(* IEC 61131-3 sources: mect_apps/TPAC1008_02_AF/Local_IO_PLC, 2 files *)

(* ---- ifTST_readVAL_writePLC.st ---- *)
(*[[
]]*)
FUNCTION ifTST_readVAL_writePLC
#import "Crosstable.gvl"
VAR_INPUT
	substatus : uint;
END_VAR

	if substatus = 0 then

		if (TST_DigIn_1 ) then RES_DigIn_1 := 0; end_if;
	    if (TST_DigIn_2 ) then RES_DigIn_2 := 0; end_if;
	    if (TST_DigIn_3 ) then RES_DigIn_3 := 0; end_if;
	    if (TST_DigIn_4 ) then RES_DigIn_4 := 0; end_if;
	    if (TST_DigIn_5 ) then RES_DigIn_5 := 0; end_if;
	    if (TST_DigIn_6 ) then RES_DigIn_6 := 0; end_if;
	    if (TST_DigIn_7 ) then RES_DigIn_7 := 0; end_if;
	    if (TST_DigIn_8 ) then RES_DigIn_8 := 0; end_if;

	    if (TST_DigOut_1) then PLC_DigOut_1 := VAL_DigOut_1; end_if;
	    if (TST_DigOut_2) then PLC_DigOut_2 := VAL_DigOut_2; end_if;
	    if (TST_DigOut_3) then PLC_DigOut_3 := VAL_DigOut_3; end_if;
	    if (TST_DigOut_4) then PLC_DigOut_4 := VAL_DigOut_4; end_if;
	    if (TST_DigOut_5) then PLC_DigOut_5 := VAL_DigOut_5; end_if;
	    if (TST_DigOut_6) then PLC_DigOut_6 := VAL_DigOut_6; end_if;
	    if (TST_DigOut_7) then PLC_DigOut_7 := VAL_DigOut_7; end_if;
	    if (TST_DigOut_8) then PLC_DigOut_8 := VAL_DigOut_8; end_if;
		if (TST_DigOut_9) then PLC_DigOut_9 := VAL_DigOut_9; end_if;
	    if (TST_DigOut_10) then PLC_DigOut_10 := VAL_DigOut_10; end_if;
	    if (TST_DigOut_11) then PLC_DigOut_11 := VAL_DigOut_11; end_if;
	    if (TST_DigOut_12) then PLC_DigOut_12 := VAL_DigOut_12; end_if;

		if (TST_AnIn_1  ) then PLC_AnInConf_1 := 0; RES_AnIn_1 := 0; end_if;
	    if (TST_AnIn_2  ) then PLC_AnInConf_2 := 0; RES_AnIn_2 := 0; end_if;
		if (TST_AnIn_3  ) then PLC_AnInConf_3 := 0; RES_AnIn_3 := 0; end_if;
	    if (TST_AnIn_4  ) then PLC_AnInConf_4 := 0; RES_AnIn_4 := 0; end_if;

	    if (TST_AnOut_1 ) then
			if (VAL_AnOutConf_1 = 3) then
				PLC_AnOutConf_1 := 2; PLC_AnOut_1 := 1000; (* 10.00 V is the PWM amplitude *)
		    else
				PLC_AnOutConf_1 := VAL_AnOutConf_1; PLC_AnOut_1 := VAL_AnOut_1;
			end_if;
		end_if;
	    if (TST_AnOut_2 ) then
			if (VAL_AnOutConf_2 = 3) then
				PLC_AnOutConf_2 := 2; PLC_AnOut_2 := 1000; (* 10.00 V is the PWM amplitude *)
		    else
				PLC_AnOutConf_2 := VAL_AnOutConf_2; PLC_AnOut_2 := VAL_AnOut_2;
			end_if;
		end_if;
		if (TST_AnOut_3 ) then
			if (VAL_AnOutConf_3 = 3) then
				PLC_AnOutConf_3 := 2; PLC_AnOut_3 := 1000; (* 10.00 V is the PWM amplitude *)
			else
				PLC_AnOutConf_3 := VAL_AnOutConf_3; PLC_AnOut_3 := VAL_AnOut_3;(* only 0..10 V *)
			end_if;
		end_if;
	    if (TST_AnOut_4) then (* only 4..20 mA *)
			PLC_AnOutConf_4 := VAL_AnOutConf_4; PLC_AnOut_4 := VAL_AnOut_4;
		end_if;

	    if (TST_Tamb      ) then RES_Tamb := 0; end_if;
		if (TST_RPM		  ) then RES_RPM := 0; end_if;

		if (TST_RTU1_WR   ) then RTU_RTU_WR := VAL_RTU1_WR; end_if;
		if (TST_RTU1_RD   ) then RES_RTU1_RD := 0; end_if;

	elsif substatus = 1 then

	    if (TST_AnOut_1 ) then
			if (VAL_AnOutConf_1 = 3) then
				PLC_AnOutConf_1 := 3; PLC_AnOut_1 := VAL_AnOut_1; (* [%] PWM *)
			end_if;
		end_if;
	    if (TST_AnOut_2 ) then
			if (VAL_AnOutConf_2 = 3) then
				PLC_AnOutConf_2 := 3; PLC_AnOut_2 := VAL_AnOut_2; (* [%] PWM *)
			end_if;
		end_if;
		if (TST_AnOut_3 ) then
			if (VAL_AnOutConf_3 = 3) then
				PLC_AnOutConf_3 := 3; PLC_AnOut_3 := VAL_AnOut_3; (* [%] PWM *)
			end_if;
		end_if;

	elsif substatus = 2 then

		if (TST_AnIn_1  ) then PLC_AnInConf_1 := VAL_AnInConf_1; end_if;
	    if (TST_AnIn_2  ) then PLC_AnInConf_2 := VAL_AnInConf_2; end_if;
		if (TST_AnIn_3  ) then PLC_AnInConf_3 := VAL_AnInConf_3; end_if;
	    if (TST_AnIn_4  ) then PLC_AnInConf_4 := VAL_AnInConf_4; end_if;

	end_if;

END_FUNCTION

(* ---- Fast.st ---- *)
(*[[
]]*)
PROGRAM Fast
#import "Crosstable.gvl"
VAR
END_VAR

;
END_PROGRAM
